// TIA Portal V16 export
// export: Created 2022-02-04T14:40:09.3980217Z, ExportSetting WithDefaults, DisplayName Totally Integrated Automation Portal, DisplayVersion V16 Update 1, DisplayName TIA Portal Version Control Interface, DisplayVersion V16, DisplayName TIA Portal Openness, DisplayVersion V16, DisplayName SINAMICS Startdrive Advanced, DisplayVersion V16 Update 5, DisplayName SINAMICS Startdrive G130, G150, S120, S150, SINAMICS MV, S210, DisplayVersion V16 Update 5, DisplayName SINAMICS Startdrive G110M, G120, G120C, G120D, G120P, G115D, DisplayVersion V16 Update 5, DisplayName STEP 7 Professional, DisplayVersion V16, DisplayName STEP 7 Safety, DisplayVersion V16, DisplayName WinCC Advanced, DisplayVersion V16, DisplayName SIMATIC Visualization Architect, DisplayVersion V16
ORGANIZATION_BLOCK "COMM_FLT"   // OB87, LAD, CommunicationError
TITLE = "Communication Fault"
VERSION : 0.1
// stored: IsIECCheckEnabled false
   VAR_TEMP
      OB87_EV_CLASS : Byte;   // 16#39 Event class 3
      OB87_FLT_ID : Byte;   // 16#XX, Fault identifcation code
      OB87_PRIORITY : Byte;   // Priority of OB Execution
      OB87_OB_NUMBR : Byte;   // 87 (Organization block 87, OB87)
      OB87_RESERVED_1 : Byte;   // Reserved for system
      OB87_RESERVED_2 : Byte;   // Reserved for system
      OB87_RESERVED_3 : Word;   // Reserved for system
      OB87_RESERVED_4 : DWord;   // Reserved for system
      OB87_DATE_TIME : Date_And_Time;   // Date and time OB87 started
   END_VAR
BEGIN
END_ORGANIZATION_BLOCK
